// TIA Portal V19 export
TYPE "User_data_type_1"
   STRUCT
      Start : Bool;
      Stop : Bool;
   END_STRUCT;
END_TYPE
